RoboDK station: ABB_irb140_Pick_and_Place.rdk

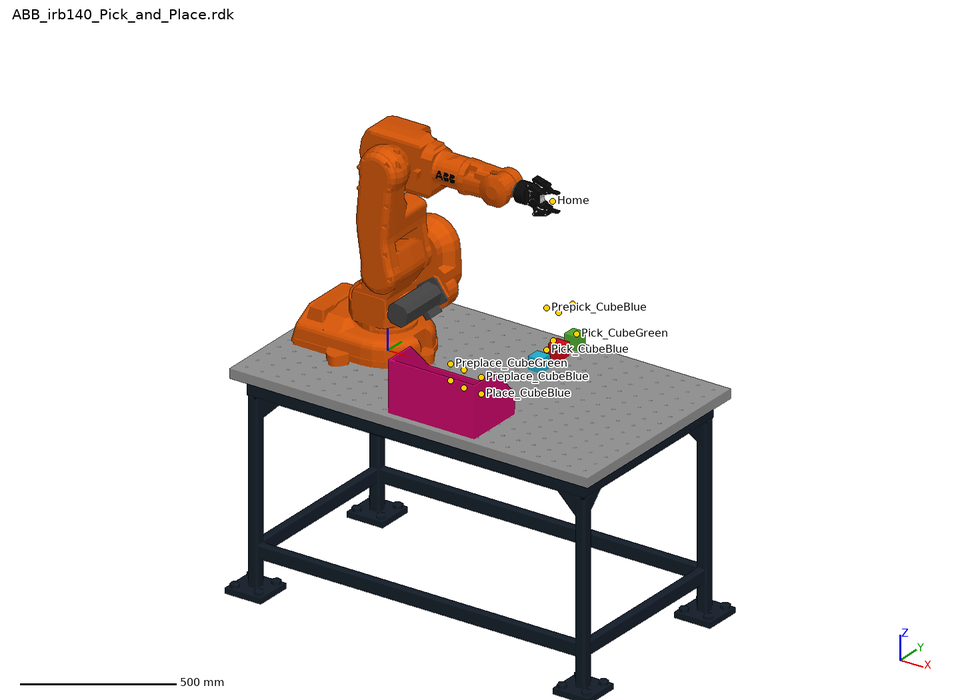
[picture v0: the station drawn from its stored meshes, robots at their saved joint values, targets as dots, program paths as lines]
Station Pick_and_Place_ABB (saved by RoboDK 5.5.4). Poses are relative to the parent item; angles as X-Y-Z fixed-axis rotations.
  - frame ABB IRB 140-6/0.8 Base at (0, 0, 0) mm
    - robot ABB IRB 140-6/0.8: 6 axes, payload 6 kg, reach 810 mm, repeatability 0.03 mm, weight 98 kg
        modified DH rows (alpha deg, a mm, theta deg, d mm): 0, 0, 0, 352; -90, 70, -90, 0; 0, 360, 0, 0; -90, 0, 0, 380; 90, 0, 0, 0; -90, 0, 180, 65
        joint limits [-180, -90, -230, -200, -120, -400] to [180, 110, 50, 200, 120, 400]; home [0, 0, 0, 0, 0, 0]; saved at [0, 0, 0, 0, 0, 0]
      - tool Gripper Closed, TCP at (0, 0, 130) mm, size 134.4 x 75 x 157.6 mm
    - target Home (Cartesian target) at (645, 0, 712) mm, rotated rx 0 ry 90 rz 0 deg; joints [0, 0, 0, 0, 0, 0] of ABB IRB 140-6/0.8
    - target Prepick_CubeBlue (Cartesian target) at (495, 180, 217) mm, rotated rx -170.72 ry -0.67 rz 106.86 deg; joints [19.578, 33.127, 6.832, 1.273, 59.289, 91.928] of ABB IRB 140-6/0.8
    - target Pick_CubeBlue (Cartesian target) at (495, 180, 67) mm, rotated rx -170.72 ry -0.67 rz 106.86 deg; joints [19.578, 51.169, 5.722, 1.624, 42.363, 91.378] of ABB IRB 140-6/0.8
    - target Preplace_CubeBlue (Cartesian target) at (525, -230, 142) mm, rotated rx -179.67 ry -0.31 rz 80.43 deg; joints [-23.732, 43.025, 4.035, 0.319, 43.332, 75.601] of ABB IRB 140-6/0.8
    - target Place_CubeBlue (Cartesian target) at (525, -230, 82) mm, rotated rx -179.67 ry -0.31 rz 80.43 deg; joints [-23.732, 50.377, 2.902, 0.363, 37.113, 75.544] of ABB IRB 140-6/0.8
    - target Prepick_CubeRed (Cartesian target) at (470.68, 279.41, 153.41) mm, rotated rx -170.86 ry 1.75 rz 92.05 deg; joints [29.733, 42.327, 3.447, 3.374, 53.183, 115.588] of ABB IRB 140-6/0.8
    - target Pick_CubeRed (Cartesian target) at (454.12, 275.65, 49.79) mm, rotated rx -170.86 ry 1.75 rz 92.05 deg; joints [30.238, 53.764, 4.326, 4.248, 40.873, 114.896] of ABB IRB 140-6/0.8
    - target Preplace_CubeRed (Cartesian target) at (451.04, -217.54, 142.43) mm, rotated rx -179.67 ry -0.31 rz 80.43 deg; joints [-25.827, 35.503, 18.554, 0.345, 36.342, 73.46] of ABB IRB 140-6/0.8
    - target Place_CubeRed (Cartesian target) at (450.74, -217.13, 77.43) mm, rotated rx -179.67 ry -0.31 rz 80.43 deg; joints [-25.801, 44.696, 17.293, 0.43, 28.411, 73.386] of ABB IRB 140-6/0.8
    - target Prepick_CubeGreen (Cartesian target) at (467.64, 364.32, 150.82) mm, rotated rx -179.61 ry 1.75 rz 92.05 deg; joints [38.308, 44.595, -0.874, -1.596, 47.642, 127.352] of ABB IRB 140-6/0.8
    - target Pick_CubeGreen (Cartesian target) at (481.85, 366.62, 45.61) mm, rotated rx -179.61 ry 1.75 rz 92.05 deg; joints [37.65, 58.429, -6.301, -1.889, 39.225, 127.083] of ABB IRB 140-6/0.8
    - target Preplace_CubeGreen (Cartesian target) at (391.88, -207.57, 142.77) mm, rotated rx -179.67 ry -0.31 rz 80.43 deg; joints [-27.992, 29.962, 29.155, 0.364, 31.289, 71.262] of ABB IRB 140-6/0.8
    - target Place_CubeGreen (Cartesian target) at (391.6, -207.19, 82.77) mm, rotated rx -179.67 ry -0.31 rz 80.43 deg; joints [-27.967, 39.658, 27.966, 0.489, 22.783, 71.148] of ABB IRB 140-6/0.8
  - program Attach Cube Blue (1 instructions, listed below)
  - program Detach Cube Blue (1 instructions, listed below)
  - program Attach Cube Red (1 instructions, listed below)
  - program Detach Cube Red (1 instructions, listed below)
  - program Attach Cube Green (1 instructions, listed below)
  - program Detach Cube Green (1 instructions, listed below)
  - frame Table_and_Bin at (0, 0, 0) mm
    - object Bin Pink at (600, -150, 0) mm, rotated rx 0 ry 0 rz 90 deg, size 225 x 337.5 x 191.2 mm, geometry from Bin-Pink.sld
    - object Table 1400x800x800mm at (0, 0, 0) mm, size 1420 x 820 x 800 mm, geometry from Table-1400x800x800mm.sld
  - Python program Pick_and_Place (listed below)
  - object Cube Blue at (450, 140, 0) mm, size 50 x 50 x 50 mm, geometry from Cube-50mm.sld
  - object Cube Red at (450, 250, 0) mm, size 50 x 50 x 50 mm, geometry from Cube-50mm.sld
  - object Cube Green at (450, 340, 0) mm, size 50 x 50 x 50 mm, geometry from Cube-50mm.sld

--- program Attach Cube Blue (robot ABB IRB 140-6/0.8) ---
  Attach to Gripper Closed

--- program Detach Cube Blue (robot ABB IRB 140-6/0.8) ---
  Detach from Gripper Closed

--- program Attach Cube Red (robot ABB IRB 140-6/0.8) ---
  Attach to Gripper Closed

--- program Detach Cube Red (robot ABB IRB 140-6/0.8) ---
  Detach from Gripper Closed

--- program Attach Cube Green (robot ABB IRB 140-6/0.8) ---
  Attach to Gripper Closed

--- program Detach Cube Green (robot ABB IRB 140-6/0.8) ---
  Detach from Gripper Closed

--- Python program Pick_and_Place ---
from robodk import robolink, robomath

# Conexión con RoboDK
RDK = robolink.Robolink()

# Obtener el robot
robot = RDK.Item('ABB IRB 140', robolink.ITEM_TYPE_ROBOT)

# Definición de la Herramienta (Gripper)
tool = RDK.Item('Gripper Closed', robolink.ITEM_TYPE_TOOL)
robot.setPoseTool(tool)

# Definición de los Cubos
cubeblue = RDK.Item('Cube Blue', robolink.ITEM_TYPE_OBJECT)
cubered = RDK.Item ('Cube Red', robolink.ITEM_TYPE_OBJECT)
cubegreen = RDK.Item ('Cube Green', robolink.ITEM_TYPE_OBJECT)

# Definir la Pose inicial de los cubos
cubeblue_home_pose = robomath.transl(450, 140, 0) * robomath.rotx(0) * robomath.roty(0) * robomath.rotz(0)
cubered_home_pose = robomath.transl(450, 250, 0) * robomath.rotx(0) * robomath.roty(0) * robomath.rotz(0)
cubegreen_home_pose = robomath.transl(450, 340, 0) * robomath.rotx(0) * robomath.roty(0) * robomath.rotz(0)


# Targets/ Puntos de paso a hacer
homecubeblue = RDK.Item('Home', robolink.ITEM_TYPE_TARGET)
prepickcubeblue = RDK.Item('Prepick_CubeBlue', robolink.ITEM_TYPE_TARGET)
pickcubeblue = RDK.Item('Pick_CubeBlue', robolink.ITEM_TYPE_TARGET)
preplacecubeblue = RDK.Item('Preplace_CubeBlue', robolink.ITEM_TYPE_TARGET)
placecubeblue = RDK.Item('Place_CubeBlue', robolink.ITEM_TYPE_TARGET)

homecubered = RDK.Item('Home', robolink.ITEM_TYPE_TARGET)
prepickcubered = RDK.Item('Prepick_CubeRed', robolink.ITEM_TYPE_TARGET)
pickcubered = RDK.Item('Pick_CubeRed', robolink.ITEM_TYPE_TARGET)
preplacecubered = RDK.Item('Preplace_CubeRed', robolink.ITEM_TYPE_TARGET)
placecubered = RDK.Item('Place_CubeRed', robolink.ITEM_TYPE_TARGET)

homecubegreen = RDK.Item('Home', robolink.ITEM_TYPE_TARGET)
prepickcubegreen = RDK.Item('Prepick_CubeGreen', robolink.ITEM_TYPE_TARGET)
pickcubegreen = RDK.Item('Pick_CubeGreen', robolink.ITEM_TYPE_TARGET)
preplacecubegreen = RDK.Item('Preplace_CubeGreen', robolink.ITEM_TYPE_TARGET)
placecubegreen = RDK.Item('Place_CubeGreen', robolink.ITEM_TYPE_TARGET)

# Programas de Attach/Detach de cada cubo
prog_attachcubeblue = RDK.Item('Attach Cube Blue', robolink.ITEM_TYPE_PROGRAM)
prog_detachcubeblue = RDK.Item('Detach Cube Blue', robolink.ITEM_TYPE_PROGRAM)

prog_attachcubered = RDK.Item('Attach Cube Red', robolink.ITEM_TYPE_PROGRAM)
prog_detachcubered = RDK.Item('Detach Cube Red', robolink.ITEM_TYPE_PROGRAM)

prog_attachcubegreen = RDK.Item('Attach Cube Green', robolink.ITEM_TYPE_PROGRAM)
prog_detachcubegreen = RDK.Item('Detach Cube Green', robolink.ITEM_TYPE_PROGRAM)

# --------------------------- Movimientos -----------------------------#

# --------------------------- Bloque Azul ------------------------------#
robot.MoveJ(homecubeblue)
robot.MoveJ(prepickcubeblue)
robot.MoveL(pickcubeblue)

prog_attachcubeblue.RunProgram()  #Correr programa para agarrar cubo azul

robot.MoveL(prepickcubeblue)
robot.MoveJ(preplacecubeblue)
robot.MoveL(placecubeblue)

prog_detachcubeblue.RunProgram()  # Correr programa para soltar cubo azul

robot.MoveL(preplacecubeblue)

# --------------------------- Bloque Rojo ------------------------------#
robot.MoveJ(homecubered)
robot.MoveJ(prepickcubered)
robot.MoveL(pickcubered)

prog_attachcubered.RunProgram()  # Correr programa para agarrar cubo rojo

robot.MoveL(prepickcubered)
robot.MoveJ(preplacecubered)
robot.MoveL(placecubered)

prog_detachcubered.RunProgram()  # Correr programa para soltar cubo rojo


robot.MoveL(preplacecubered)

# --------------------------- Bloque Verde ------------------------------#
robot.MoveJ(homecubegreen)
robot.MoveJ(prepickcubegreen)
robot.MoveL(pickcubegreen)

prog_attachcubegreen.RunProgram()  # Correr programa para agarrar cubo verde

robot.MoveL(prepickcubegreen)
robot.MoveJ(preplacecubegreen)
robot.MoveL(placecubegreen)

prog_detachcubegreen.RunProgram()  # Correr programa para soltar cubo verde

robot.MoveL(preplacecubered)

# Regresar a home
robot.MoveJ(homecubeblue)

# ----- Poner el cubo a su lugar -----
cubeblue.setPoseAbs(cubeblue_home_pose)
cubered.setPoseAbs(cubered_home_pose)
cubegreen.setPoseAbs(cubegreen_home_pose)

#print("✔️ Secuencia completada y cubo restablecido a posición original.")
